(* IEC 61131-3 sources: tipps-and-tricks/src, 3 files *)

(* ---- Code.st ---- *)
NAMESPACE Simatic.Ax

    {axcode:docs-v0:@simatic-ax/tipps_and_tricks:app.md}
    CLASS Code
        VAR
            test : INT := 3;
            myBool : BOOL;
        END_VAR

        /// Block description:
        /// here i can write my comment
        /// Return value:
        METHOD Name : INT
            VAR_INPUT // here i can put my comments
            END_VAR
            IF (TRUE) THEN
                 myBool := TRUE;
            END_IF;
        END_METHOD
    END_CLASS

END_NAMESPACE

(* ---- Configuration.st ---- *)
CONFIGURATION PLC_1
    TASK Main(Interval := T#1000ms, Priority := 1);
    PROGRAM P1 WITH Main : SampleProgram;
    VAR_GLOBAL
        newname1 : DINT; // former of type BOOL
        newname2 : DINT; // former of type BOOL
    END_VAR
END_CONFIGURATION

PROGRAM SampleProgram
    VAR_EXTERNAL
        newname1 : DINT; // former of type BOOL
        newname2 : DINT; // former of type BOOL
    END_VAR
    VAR

    END_VAR

    ;
END_PROGRAM

(* ---- MainProgram.st ---- *)
PROGRAM MainProgram
    VAR_EXTERNAL
    END_VAR

    VAR
    END_VAR

    VAR_TEMP
    END_VAR
    ;
END_PROGRAM
